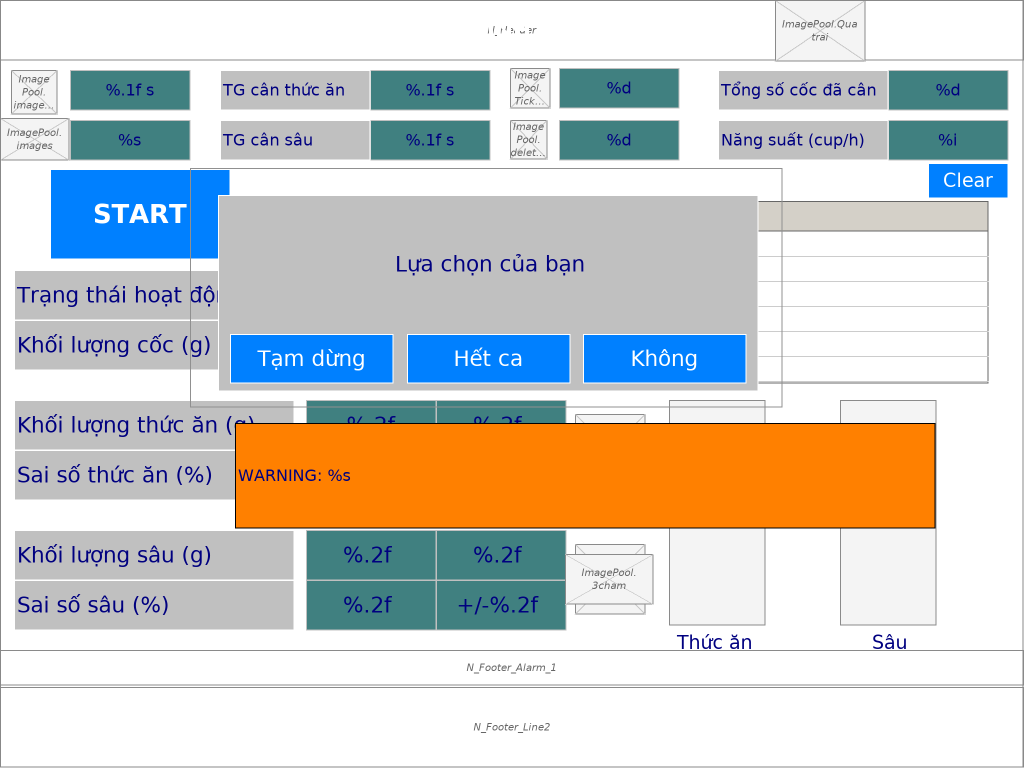
VISUALIZATION MAIN_LINE2  // 1024x768
    Rectangle (49,168 180x90), "STOP", invisible if: not bStatusStart2, input disabled if: not bStatusStart2
        OnMouseDown: execute { hienthiDialog2 := TRUE; }
    Rectangle (50,169 180x90), "START", invisible if: bStatusStart2, input disabled if: Not bRunAuto
        OnMouseDown: execute { bStart2 := true; }
    Frame (0,687 1024x80)
        shows N_Footer_Line2()
    Frame (0,0 1024x60)
        shows N_Header()
    Textfield (353,5 400x50), "MÀN HÌNH CHÍNH LINE 2"
    Rectangle (70,70 120x40), "%.1f s", text variable: PR_Line02.timeCycle
    Rectangle (370,70 120x40), "%.1f s", text variable: PR_Line02.fb_FoodWeight.fTime
    Image (11,70 46x44), image: ImagePool.images (1)
    Rectangle (70,120 120x40), "%s", text variable: PRG_MainRecipe1_1.RecipeName
    Image (0,118 69x42), image: ImagePool.images
    Rectangle (888,70 120x40), "%d", text variable: nCount2
    Image (510,68 40x40), image: ImagePool.Tick-Green-Check-Mark-PNG-Clipart
    Rectangle (559,68 120x40), "%d", text variable: nResult_true2
    Image (510,120 37x39), image: ImagePool.delete-button-png-28575
    Rectangle (559,120 120x40), "%d", text variable: nResult_false2
    Rectangle (928,163 80x35), "Clear"
        tap GVL_OF_VU.bClear[2]
        OnMouseDown: execute { bClear2 := true; }
    Rectangle (370,120 120x40), "%.1f s", text variable: PR_Line02.fb_WormWeight.fTime
    Image (775,0 90x61), image: ImagePool.Qua trai
        OnMouseClick: change screen: MAIN_LINE1
        OnMouseClick: execute { MAIN.bModeAuto := TRUE; MAIN.bModeManual := FALSE; }
    RoundedRectangle (840,625 100x35), "Sâu"
    RoundedRectangle (665,625 100x35), "Thức ăn"
    Rectangle (306,400 130x50), "%.2f", text variable: PR_Line02.fb_FoodWeight.fWeight_Food
    Rectangle (306,450 130x50), "%.2f", text variable: PR_Line02.fb_FoodWeight.fActDelta_Food
    Rectangle (306,320 260x50), "%.2f", text variable: PR_Line02.fb_FoodWeight.fTareWeight
    Rectangle (436,400 130x50), "%.2f", text variable: PR_Line02.fDerisedWeight_Food
    Rectangle (436,450 130x50), "+/-%.2f", text variable: PR_Line02.fDelta_Food
    Rectangle (306,200 130x60), "Thực tế"
    Rectangle (306,270 260x50), "%s", text variable: nStatus2
    Rectangle (437,200 130x60), "Cài đặt"
    Rectangle (306,530 130x50), "%.2f", text variable: PR_Line02.fb_WormWeight.fWeight_Worm
    Rectangle (306,580 130x50), "%.2f", text variable: PR_Line02.fb_WormWeight.fActDelta_Worm
    Rectangle (436,530 130x50), "%.2f", text variable: PR_Line02.fDerisedWeight_Worm
    Rectangle (436,580 130x50), "+/-%.2f", text variable: PR_Line02.fDelta_Worm
    BarDisplayImage (669,400 96x225), value: PR_Line02.fb_FoodWeight.fWeight_Food, style: BarDisplayImage-Gray, scale format: %.1f, scale 0..18
    BarDisplayImage (840,400 96x225), value: PR_Line02.fb_WormWeight.fWeight_Worm, style: BarDisplayImage-Gray, scale format: %.1f, scale 0..5
    Rectangle (14,270 280x50), "Trạng thái hoạt động"
    Rectangle (14,530 280x50), "Khối lượng sâu (g)"
    Rectangle (14,580 280x50), "Sai số sâu (%)"
    Rectangle (14,320 280x50), "Khối lượng cốc (g)"
    Rectangle (14,450 280x50), "Sai số thức ăn (%)"
    Rectangle (14,400 280x50), "Khối lượng thức ăn (g)"
    ImageSwitcher (575,414 70x70), variable: PR_Line02.fb_FoodWeight.bStatus_Food, invisible if: not PR_Line02.fb_FoodWeight.bStatus, input disabled if: true, background image: ImagePool.262-2627516_clipart-cross-tick-green-tick-png-icon, image: ImagePool.delete-button-png-28575, behaviour: TOGGLE
    ImageSwitcher (575,544 70x70), variable: PR_Line02.fb_WormWeight.bStatus_Worm, invisible if: not PR_Line02.fb_WormWeight.bStatus, input disabled if: true, background image: ImagePool.262-2627516_clipart-cross-tick-green-tick-png-icon, image: ImagePool.delete-button-png-28575, behaviour: TOGGLE
    Table (615,201 373x182), data array: PR_Line02.fProductLog
        p3854506369: PR_Line02.fProductLog[1][INDEX]
        p1892666644: PR_Line02.fProductLog[2][INDEX]
        p2232123230: Thức ăn
        p511219082: Sâu
    Frame (0,650 1024x35)
        shows N_Footer_Alarm_1()
    Rectangle (888,120 120x40), "%i", text variable: PR_Line02.fproduct
    Rectangle (718,70 170x40), "Tổng số cốc đã cân"
    Rectangle (220,70 150x40), "TG cân thức ăn"
    Rectangle (220,120 150x40), "TG cân sâu"
    Rectangle (718,120 170x40), "Năng suất (cup/h)"
    Image (565,554 88x50), invisible if: PR_Line02.fb_WormWeight.bStatus, image: ImagePool.3cham
    Image (565,424 88x50), invisible if: PR_Line02.fb_FoodWeight.bStatus, image: ImagePool.3cham
    GroupBox (190,160 592x247), invisible if: not hienthiDialog2, input disabled if: not hienthiDialog2
        Rectangle (28,35 540x196), invisible if: not hienthiDialog2, input disabled if: not hienthiDialog2
        Rectangle (393,174 163x49), "Không", invisible if: not hienthiDialog2, input disabled if: not hienthiDialog2
            OnMouseDown: execute { hienthiDialog2 := FALSE; }
        Label (107,78 386x52), "Lựa chọn của bạn", invisible if: not hienthiDialog
        Rectangle (40,174 163x49), "Tạm dừng", input disabled if: not hienthiDialog2
            OnMouseDown: execute { bStop2 := TRUE; hienthiDialog2 := FALSE; }
        Rectangle (217,174 163x49), "Hết ca", invisible if: not hienthiDialog2, input disabled if: not hienthiDialog2
            OnMouseDown: execute { bShift_is_over2 := TRUE; hienthiDialog2 := FALSE; }
    Rectangle (235,423 700x105), "WARNING: %s", text variable: StWarningTxt3, invisible if: not bAlarm_Iot, input disabled if: not bAlarm_Iot
END_VISUALIZATION

(* stored: Version 1.1.0.1, ProductVersion 3.1.4024.12
   Visu MAIN_LINE2: Id {279637b3-9929-4464-87af-ca2aa9556ae6} *)
